FUNCTION Grip : INT
VAR_INPUT
	EndPosition: INT;
	State: INT;
END_VAR
VAR
	MovementEnum: Movement;
	NextState: INT;
	MotorDirectionEnum: MovementDirection;
END_VAR

IF Automatic.GripPositionAuto > EndPosition THEN
	MotorDirectionEnum := MovementDirection.TowardsSensor;
ELSE
	MotorDirectionEnum := MovementDirection.AwayFromSensor;
END_IF

IF MotorDirectionEnum = MovementDirection.TowardsSensor THEN
	IF Automatic.GripPositionAuto > EndPosition THEN
		IO.MotorGripDirection := (MotorDirectionEnum = MovementDirection.TowardsSensor);
		IF NOT Automatic.SafetyGON THEN
			Automatic.GCurrentlyMoving := TRUE;
			IO.MotorGrip := (MovementEnum = Movement.ON);
		END_IF
		NextState := State;
	ELSE
		IO.MotorGrip := (MovementEnum = Movement.OFF);
		NextState := State + 1;
		Automatic.GCurrentlyMoving := FALSE;
	END_IF
ELSE
	IF Automatic.GripPositionAuto < EndPosition THEN
		IO.MotorGripDirection := (MotorDirectionEnum = MovementDirection.AwayFromSensor);
		IF NOT Automatic.SafetyGON THEN
			Automatic.GCurrentlyMoving := TRUE;
			IO.MotorGrip := (MovementEnum = Movement.ON);
		END_IF
		NextState := State;
	ELSE
		IO.MotorGrip := (MovementEnum = Movement.OFF);
		NextState := State + 1;
		Automatic.GCurrentlyMoving := FALSE;
	END_IF
END_IF

Grip := NextState;
RETURN;

END_FUNCTION

(* stored: Version 1.1.0.1, ProductVersion 3.1.4024.13
   POU Grip: Id {69c52a9e-9855-458c-8351-023b987ea65f}, SpecialFunc None *)
